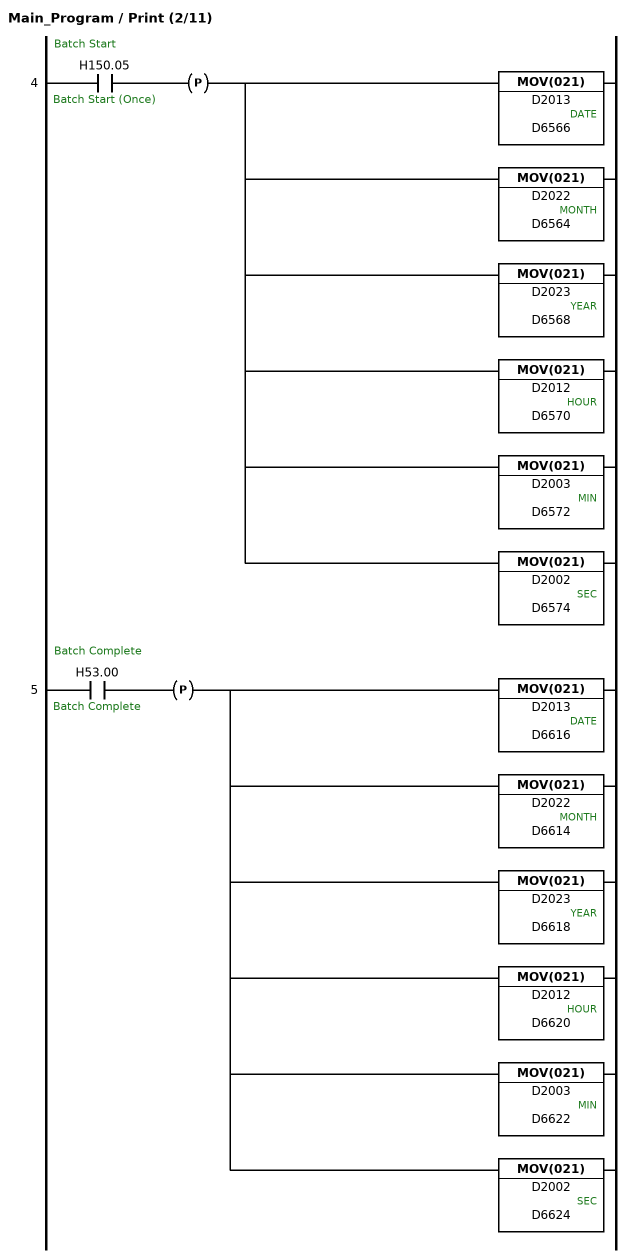
; [picture p48: Main_Program / Print, rungs 4-5]
; rung 4: Batch Start
LD H150.05  ; Batch Start (Once)
UP(521)
MOV(021) D2013 D6566  ; DATE
MOV(021) D2022 D6564  ; MONTH
MOV(021) D2023 D6568  ; YEAR
MOV(021) D2012 D6570  ; HOUR
MOV(021) D2003 D6572  ; MIN
MOV(021) D2002 D6574  ; SEC
; rung 5: Batch Complete
LD H53.00  ; Batch Complete
UP(521)
MOV(021) D2013 D6616  ; DATE
MOV(021) D2022 D6614  ; MONTH
MOV(021) D2023 D6618  ; YEAR
MOV(021) D2012 D6620  ; HOUR
MOV(021) D2003 D6622  ; MIN
MOV(021) D2002 D6624  ; SEC

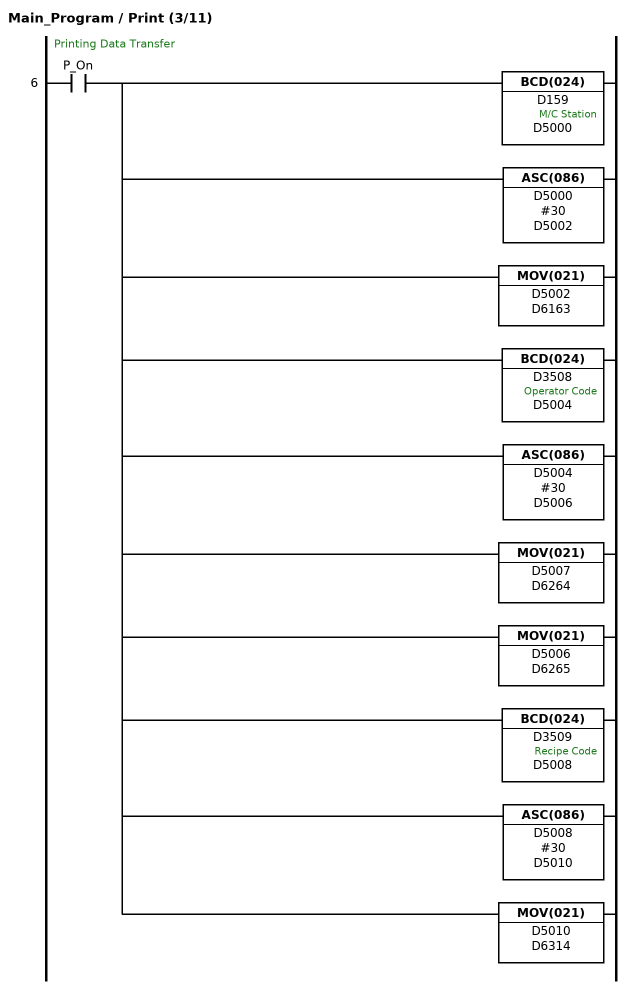
; rung 6: Printing Data Transfer
LD P_On
BCD(024) D159 D5000  ; M/C Station
ASC(086) D5000 #30 D5002
MOV(021) D5002 D6163
BCD(024) D3508 D5004  ; Operator Code
ASC(086) D5004 #30 D5006
MOV(021) D5007 D6264
MOV(021) D5006 D6265
BCD(024) D3509 D5008  ; Recipe Code
ASC(086) D5008 #30 D5010
MOV(021) D5010 D6314

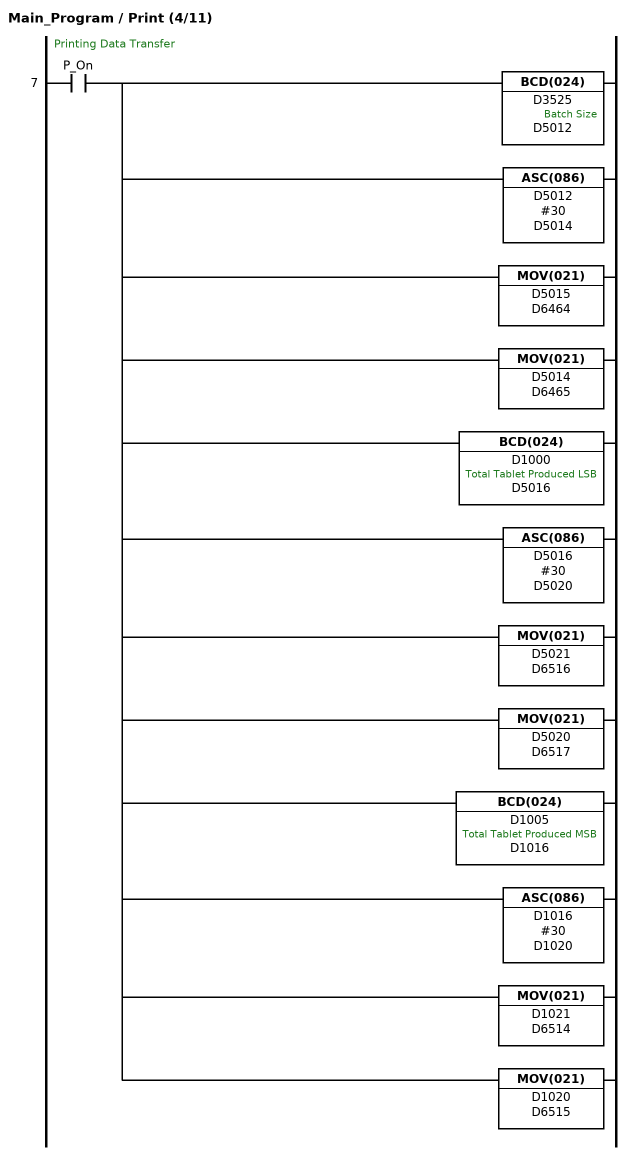
; rung 7: Printing Data Transfer
LD P_On
BCD(024) D3525 D5012  ; Batch Size
ASC(086) D5012 #30 D5014
MOV(021) D5015 D6464
MOV(021) D5014 D6465
BCD(024) D1000 D5016  ; Total Tablet Produced LSB
ASC(086) D5016 #30 D5020
MOV(021) D5021 D6516
MOV(021) D5020 D6517
BCD(024) D1005 D1016  ; Total Tablet Produced MSB
ASC(086) D1016 #30 D1020
MOV(021) D1021 D6514
MOV(021) D1020 D6515

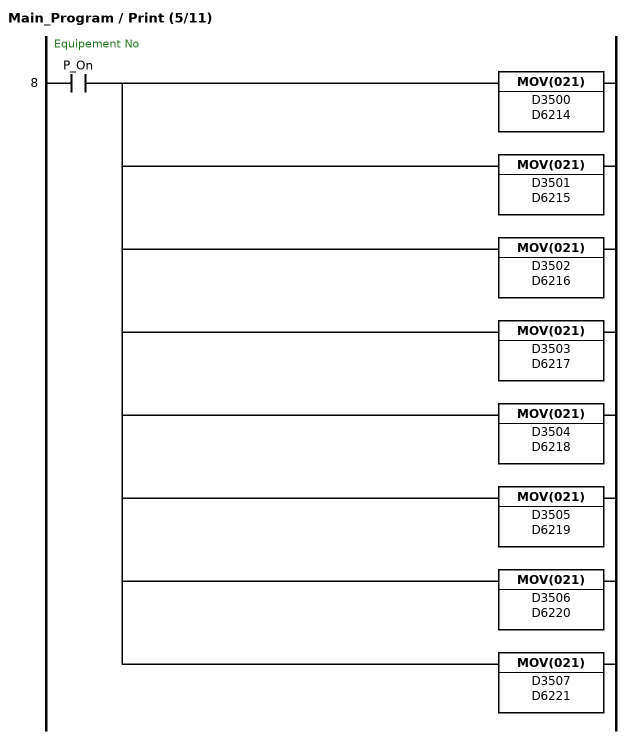
; rung 8: Equipement No
LD P_On
MOV(021) D3500 D6214
MOV(021) D3501 D6215
MOV(021) D3502 D6216
MOV(021) D3503 D6217
MOV(021) D3504 D6218
MOV(021) D3505 D6219
MOV(021) D3506 D6220
MOV(021) D3507 D6221

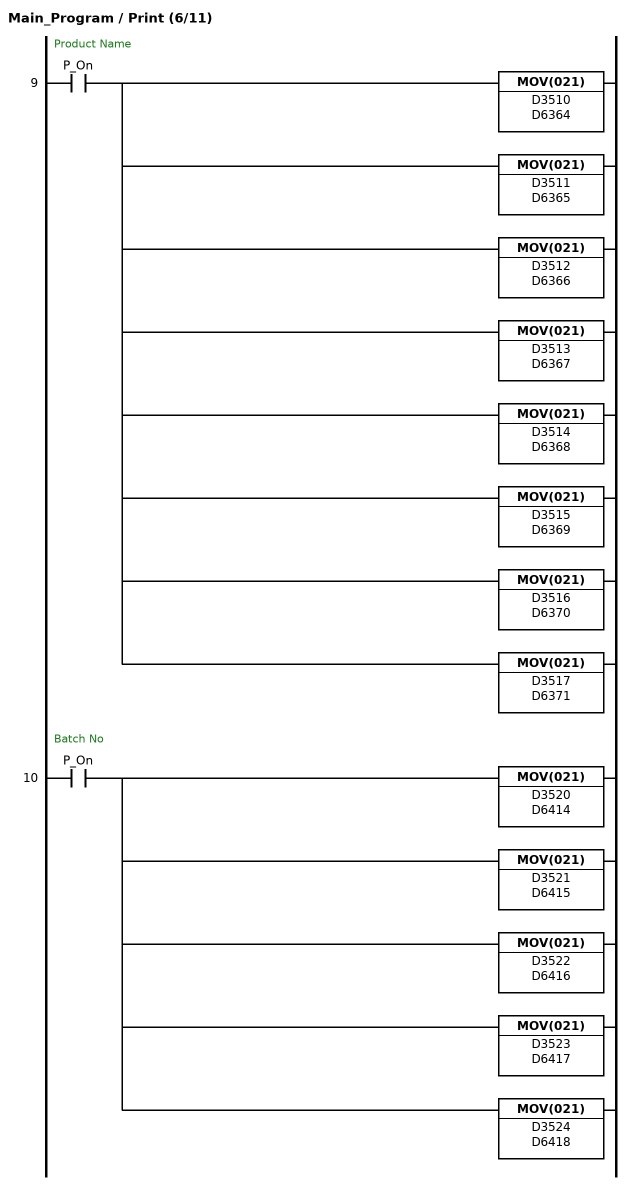
; rung 9: Product Name
LD P_On
MOV(021) D3510 D6364
MOV(021) D3511 D6365
MOV(021) D3512 D6366
MOV(021) D3513 D6367
MOV(021) D3514 D6368
MOV(021) D3515 D6369
MOV(021) D3516 D6370
MOV(021) D3517 D6371
; rung 10: Batch No
LD P_On
MOV(021) D3520 D6414
MOV(021) D3521 D6415
MOV(021) D3522 D6416
MOV(021) D3523 D6417
MOV(021) D3524 D6418

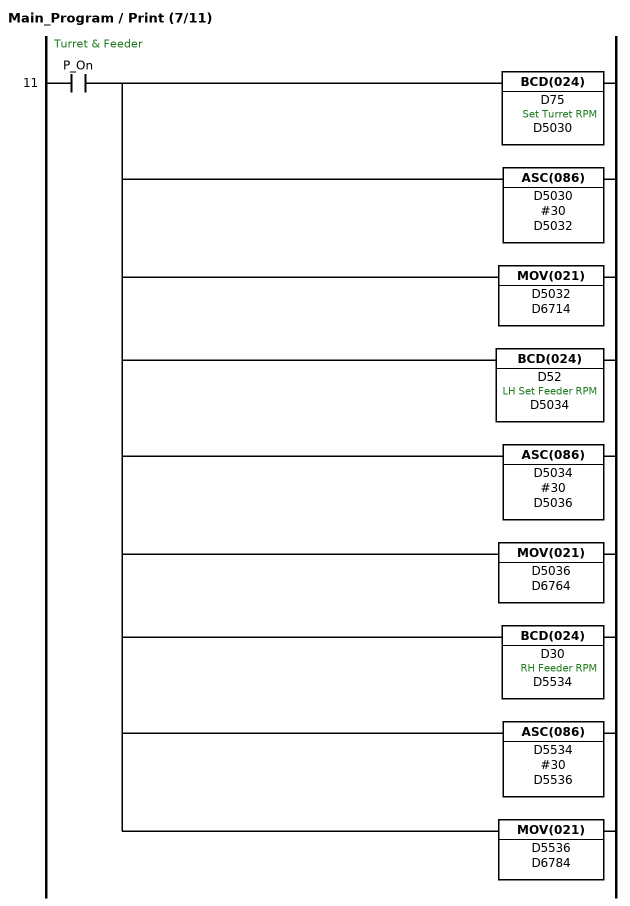
; rung 11: Turret & Feeder
LD P_On
BCD(024) D75 D5030  ; Set Turret RPM
ASC(086) D5030 #30 D5032
MOV(021) D5032 D6714
BCD(024) D52 D5034  ; LH Set Feeder RPM
ASC(086) D5034 #30 D5036
MOV(021) D5036 D6764
BCD(024) D30 D5534  ; RH Feeder RPM
ASC(086) D5534 #30 D5536
MOV(021) D5536 D6784

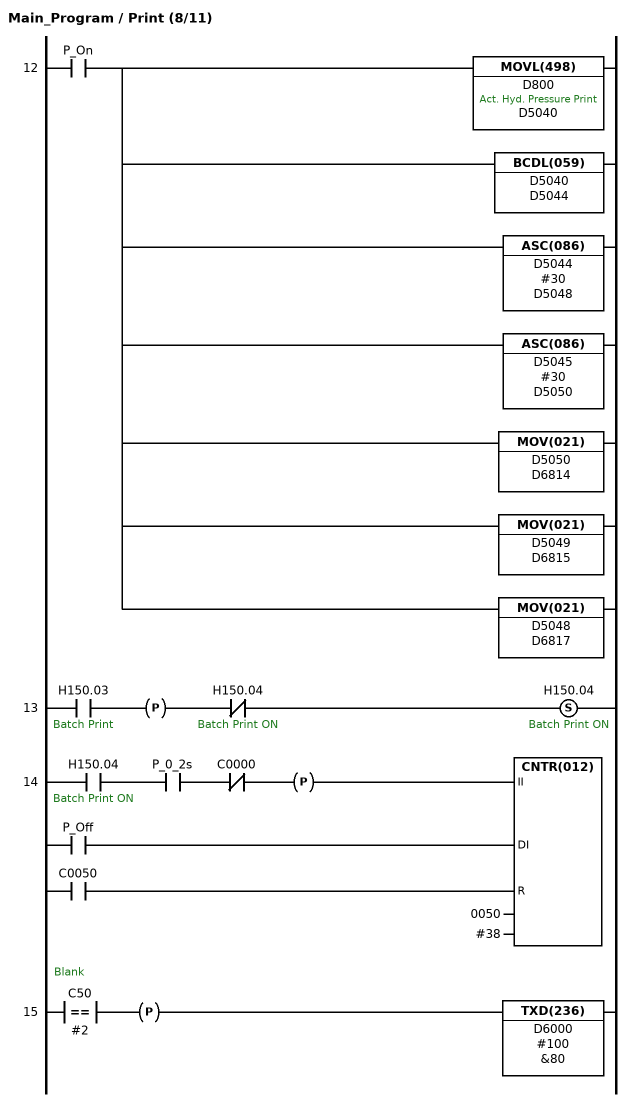
; rung 12
LD P_On
MOVL(498) D800 D5040  ; Act. Hyd. Pressure Print
BCDL(059) D5040 D5044
ASC(086) D5044 #30 D5048
ASC(086) D5045 #30 D5050
MOV(021) D5050 D6814
MOV(021) D5049 D6815
MOV(021) D5048 D6817
; rung 13
LD H150.03  ; Batch Print
UP(521)
ANDNOT H150.04  ; Batch Print ON
SET H150.04  ; Batch Print ON
; rung 14
LD H150.04  ; Batch Print ON
AND P_0_2s
ANDNOT C0000
UP(521)
LD P_Off
LD C0050
CNTR(012) 0050 #38
; rung 15: Blank
LD=(300) C50 #2
UP(521)
TXD(236) D6000 #100 &80

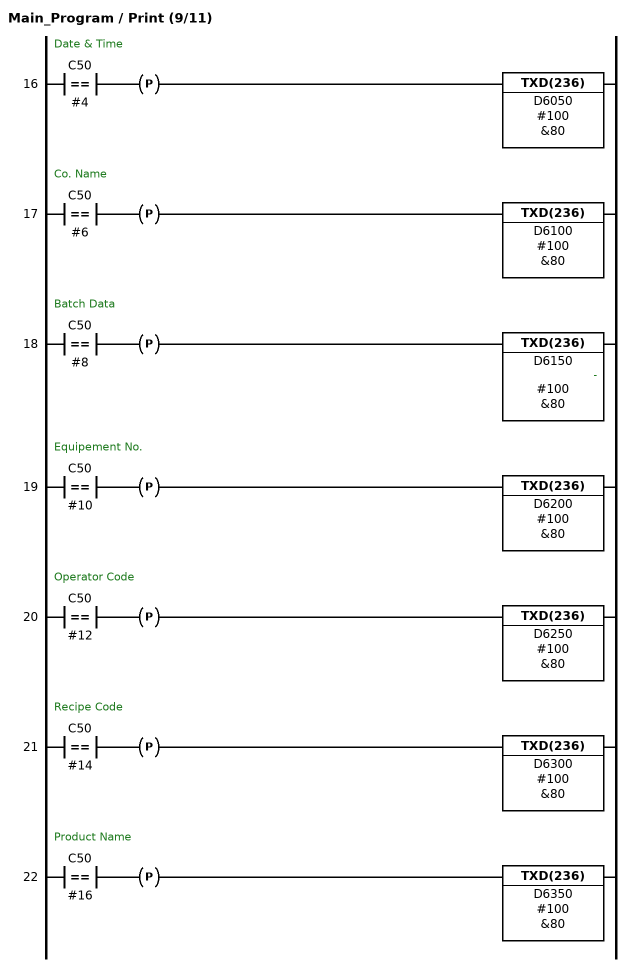
; rung 16: Date & Time
LD=(300) C50 #4
UP(521)
TXD(236) D6050 #100 &80
; rung 17: Co. Name
LD=(300) C50 #6
UP(521)
TXD(236) D6100 #100 &80
; rung 18: Batch Data
LD=(300) C50 #8
UP(521)
TXD(236) D6150 #100 &80  ; -
; rung 19: Equipement No.
LD=(300) C50 #10
UP(521)
TXD(236) D6200 #100 &80
; rung 20: Operator Code
LD=(300) C50 #12
UP(521)
TXD(236) D6250 #100 &80
; rung 21: Recipe Code
LD=(300) C50 #14
UP(521)
TXD(236) D6300 #100 &80
; rung 22: Product Name
LD=(300) C50 #16
UP(521)
TXD(236) D6350 #100 &80

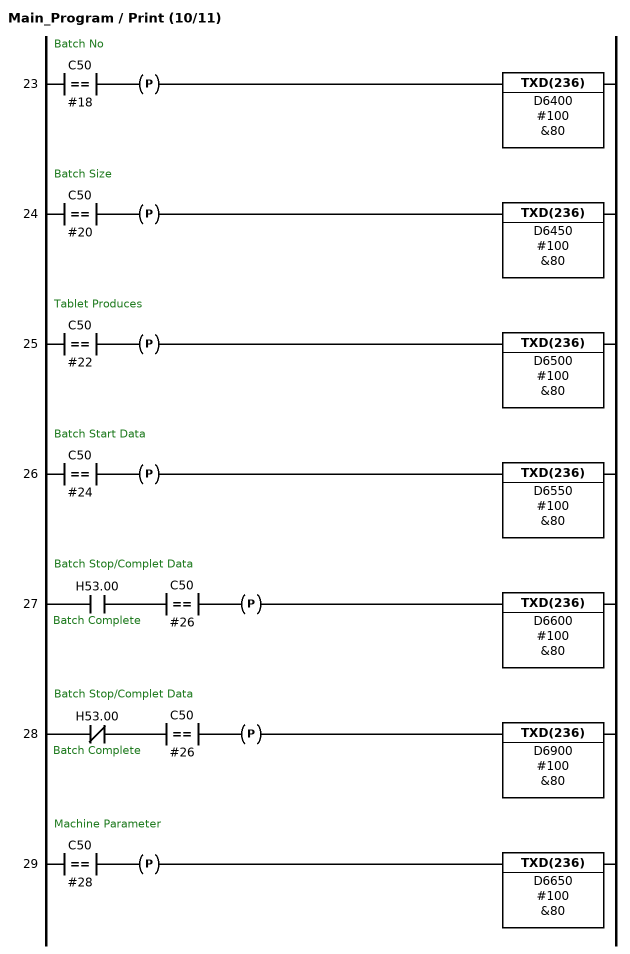
; rung 23: Batch No
LD=(300) C50 #18
UP(521)
TXD(236) D6400 #100 &80
; rung 24: Batch Size
LD=(300) C50 #20
UP(521)
TXD(236) D6450 #100 &80
; rung 25: Tablet Produces
LD=(300) C50 #22
UP(521)
TXD(236) D6500 #100 &80
; rung 26: Batch Start Data
LD=(300) C50 #24
UP(521)
TXD(236) D6550 #100 &80
; rung 27: Batch Stop/Complet Data
LD H53.00  ; Batch Complete
AND=(300) C50 #26
UP(521)
TXD(236) D6600 #100 &80
; rung 28: Batch Stop/Complet Data
LDNOT H53.00  ; Batch Complete
AND=(300) C50 #26
UP(521)
TXD(236) D6900 #100 &80
; rung 29: Machine Parameter
LD=(300) C50 #28
UP(521)
TXD(236) D6650 #100 &80

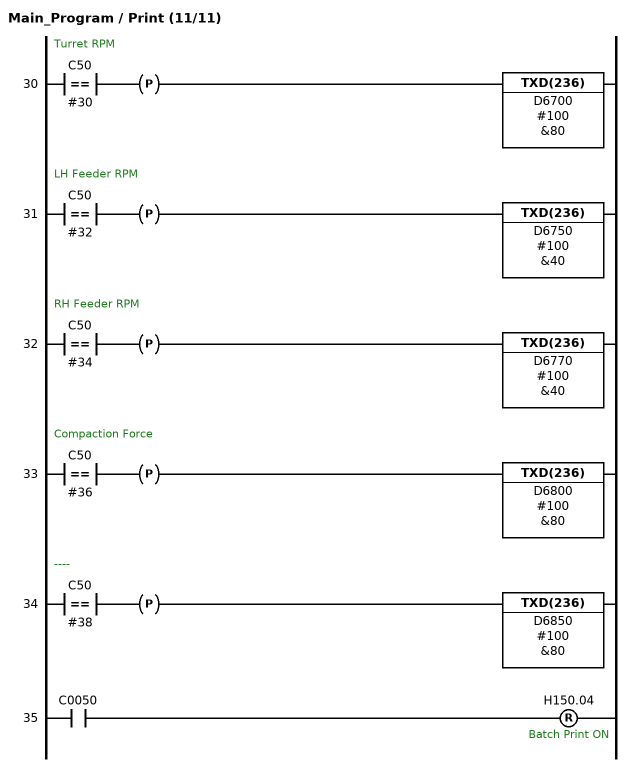
; rung 30: Turret RPM
LD=(300) C50 #30
UP(521)
TXD(236) D6700 #100 &80
; rung 31: LH Feeder RPM
LD=(300) C50 #32
UP(521)
TXD(236) D6750 #100 &40
; rung 32: RH Feeder RPM
LD=(300) C50 #34
UP(521)
TXD(236) D6770 #100 &40
; rung 33: Compaction Force
LD=(300) C50 #36
UP(521)
TXD(236) D6800 #100 &80
; rung 34: ----
LD=(300) C50 #38
UP(521)
TXD(236) D6850 #100 &80
; rung 35
LD C0050
RSET H150.04  ; Batch Print ON

### Section sampling_hooter

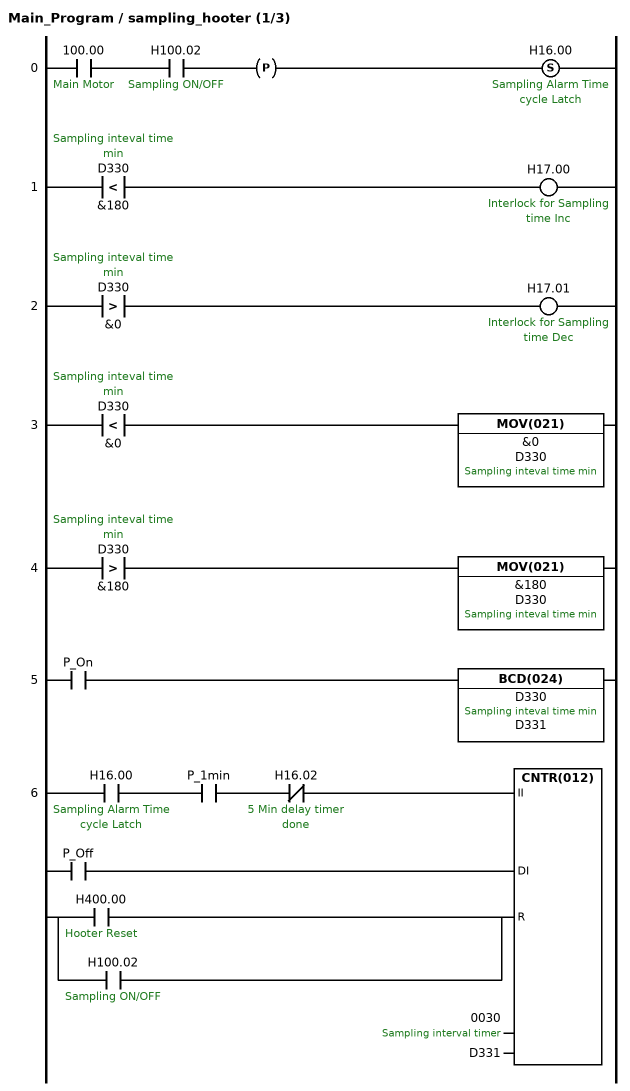
; rung 0
LD 100.00  ; Main Motor
AND H100.02  ; Sampling ON/OFF
UP(521)
SET H16.00  ; Sampling Alarm Time cycle Latch
; rung 1
LD<(310) D330 &180  ; Sampling inteval time min
OUT H17.00  ; Interlock for Sampling time Inc
; rung 2
LD>(320) D330 &0  ; Sampling inteval time min
OUT H17.01  ; Interlock for Sampling time Dec
; rung 3
LD<(310) D330 &0  ; Sampling inteval time min
MOV(021) &0 D330  ; Sampling inteval time min
; rung 4
LD>(320) D330 &180  ; Sampling inteval time min
MOV(021) &180 D330  ; Sampling inteval time min
; rung 5
LD P_On
BCD(024) D330 D331  ; Sampling inteval time min
; rung 6
LD H16.00  ; Sampling Alarm Time cycle Latch
AND P_1min
ANDNOT H16.02  ; 5 Min delay timer done
LD P_Off
LD H400.00  ; Hooter Reset
OR H100.02  ; Sampling ON/OFF
CNTR(012) 0030 D331  ; Sampling interval timer

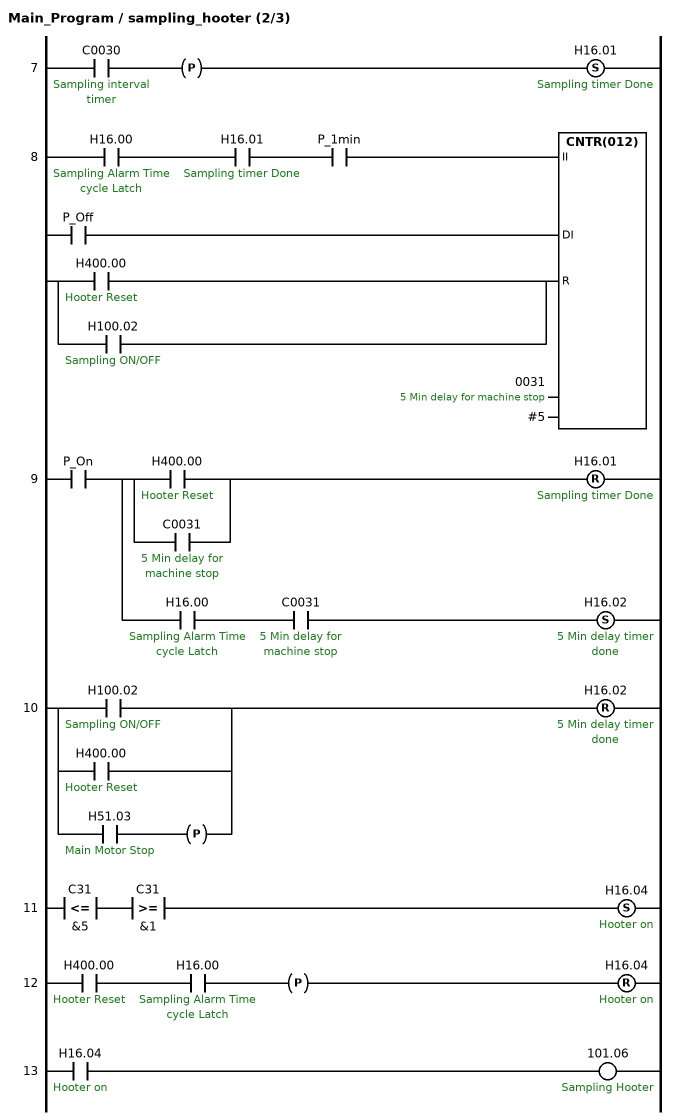
; rung 7
LD C0030  ; Sampling interval timer
UP(521)
SET H16.01  ; Sampling timer Done
; rung 8
LD H16.00  ; Sampling Alarm Time cycle Latch
AND H16.01  ; Sampling timer Done
AND P_1min
LD P_Off
LD H400.00  ; Hooter Reset
OR H100.02  ; Sampling ON/OFF
CNTR(012) 0031 #5  ; 5 Min delay for machine stop
; rung 9
LD P_On
OUT TR0
LD H400.00  ; Hooter Reset
OR C0031  ; 5 Min delay for machine stop
ANDLD
RSET H16.01  ; Sampling timer Done
LD TR0
AND H16.00  ; Sampling Alarm Time cycle Latch
AND C0031  ; 5 Min delay for machine stop
SET H16.02  ; 5 Min delay timer done
; rung 10
LD H100.02  ; Sampling ON/OFF
OR H400.00  ; Hooter Reset
LD H51.03  ; Main Motor Stop
UP(521)
ORLD
RSET H16.02  ; 5 Min delay timer done
; rung 11
LD<=(315) C31 &5
AND>=(325) C31 &1
SET H16.04  ; Hooter on
; rung 12
LD H400.00  ; Hooter Reset
AND H16.00  ; Sampling Alarm Time cycle Latch
UP(521)
RSET H16.04  ; Hooter on
; rung 13
LD H16.04  ; Hooter on
OUT 101.06  ; Sampling Hooter

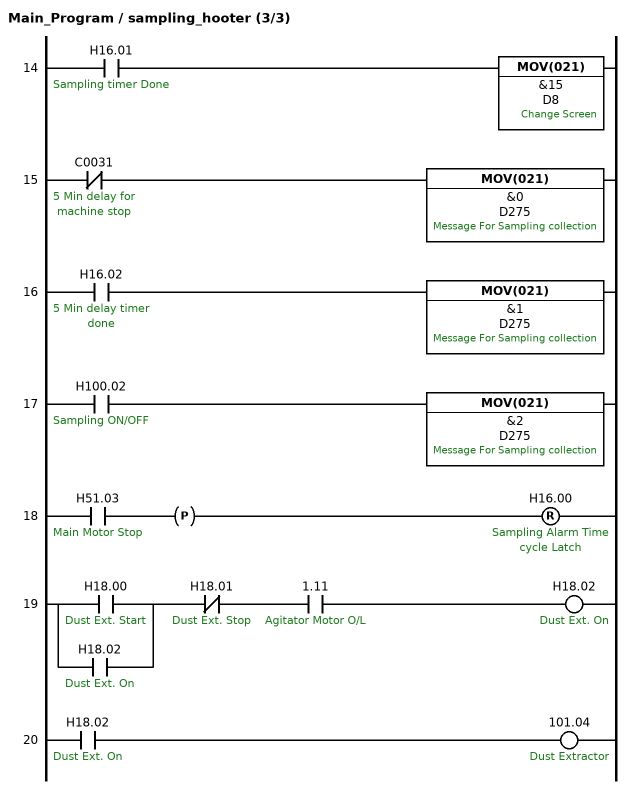
; rung 14
LD H16.01  ; Sampling timer Done
MOV(021) &15 D8  ; Change Screen
; rung 15
LDNOT C0031  ; 5 Min delay for machine stop
MOV(021) &0 D275  ; Message For Sampling collection
; rung 16
LD H16.02  ; 5 Min delay timer done
MOV(021) &1 D275  ; Message For Sampling collection
; rung 17
LD H100.02  ; Sampling ON/OFF
MOV(021) &2 D275  ; Message For Sampling collection
; rung 18
LD H51.03  ; Main Motor Stop
UP(521)
RSET H16.00  ; Sampling Alarm Time cycle Latch
; rung 19
LD H18.00  ; Dust Ext. Start
OR H18.02  ; Dust Ext. On
ANDNOT H18.01  ; Dust Ext. Stop
AND 1.11  ; Agitator Motor O/L
OUT H18.02  ; Dust Ext. On
; rung 20
LD H18.02  ; Dust Ext. On
OUT 101.04  ; Dust Extractor

### Section Vac_U_Max

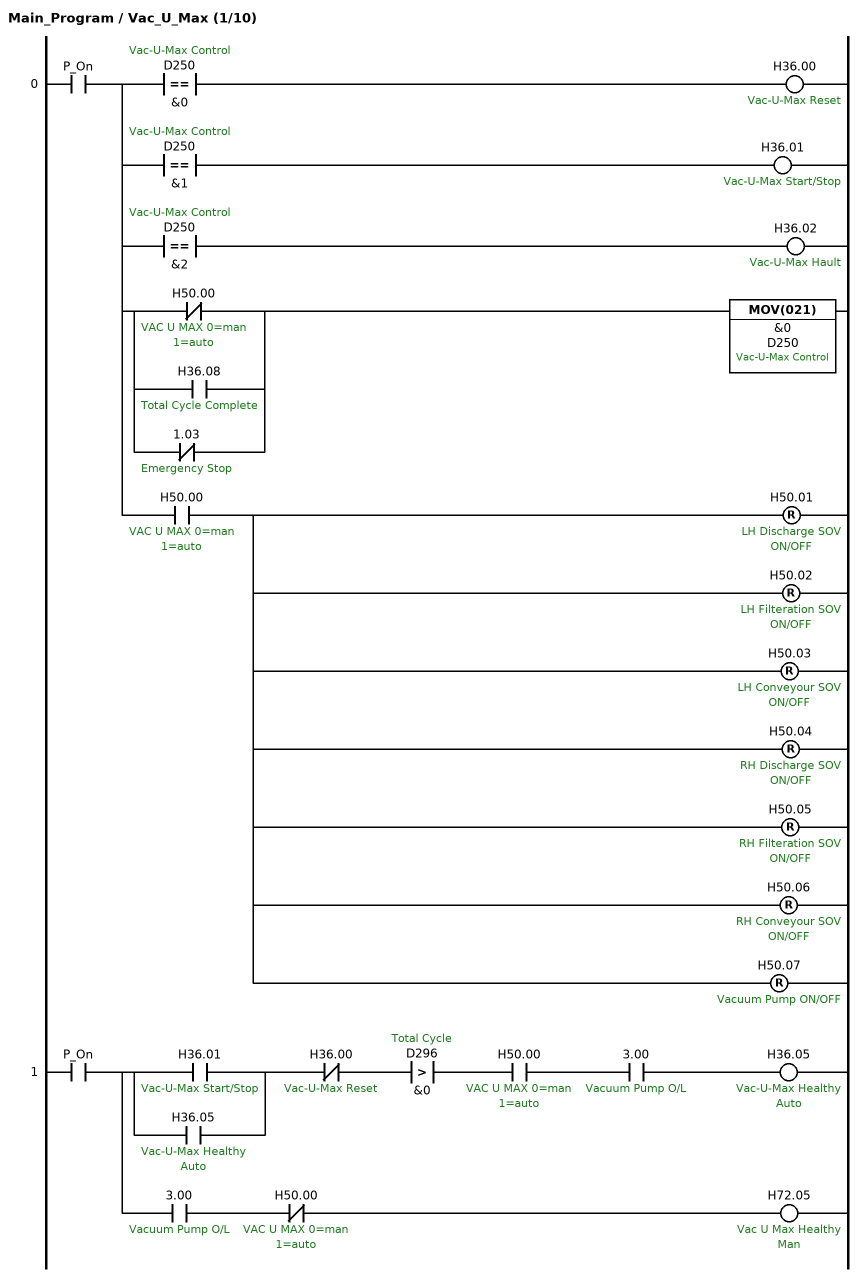
; rung 0
LD P_On
OUT TR0
AND=(300) D250 &0  ; Vac-U-Max Control
OUT H36.00  ; Vac-U-Max Reset
LD TR0
AND=(300) D250 &1  ; Vac-U-Max Control
OUT H36.01  ; Vac-U-Max Start/Stop
LD TR0
AND=(300) D250 &2  ; Vac-U-Max Control
OUT H36.02  ; Vac-U-Max Hault
LD TR0
LDNOT H50.00  ; VAC U MAX 0=man 1=auto
OR H36.08  ; Total Cycle Complete
ORNOT 1.03  ; Emergency Stop
ANDLD
MOV(021) &0 D250  ; Vac-U-Max Control
LD TR0
AND H50.00  ; VAC U MAX 0=man 1=auto
RSET H50.01  ; LH Discharge SOV ON/OFF
RSET H50.02  ; LH Filteration SOV ON/OFF
RSET H50.03  ; LH Conveyour SOV ON/OFF
RSET H50.04  ; RH Discharge SOV ON/OFF
RSET H50.05  ; RH Filteration SOV ON/OFF
RSET H50.06  ; RH Conveyour SOV ON/OFF
RSET H50.07  ; Vacuum Pump ON/OFF
; rung 1
LD P_On
OUT TR0
LD H36.01  ; Vac-U-Max Start/Stop
OR H36.05  ; Vac-U-Max Healthy Auto
ANDLD
ANDNOT H36.00  ; Vac-U-Max Reset
AND>(320) D296 &0  ; Total Cycle
AND H50.00  ; VAC U MAX 0=man 1=auto
AND 3.00  ; Vacuum Pump O/L
OUT H36.05  ; Vac-U-Max Healthy Auto
LD TR0
AND 3.00  ; Vacuum Pump O/L
ANDNOT H50.00  ; VAC U MAX 0=man 1=auto
OUT H72.05  ; Vac U Max Healthy Man

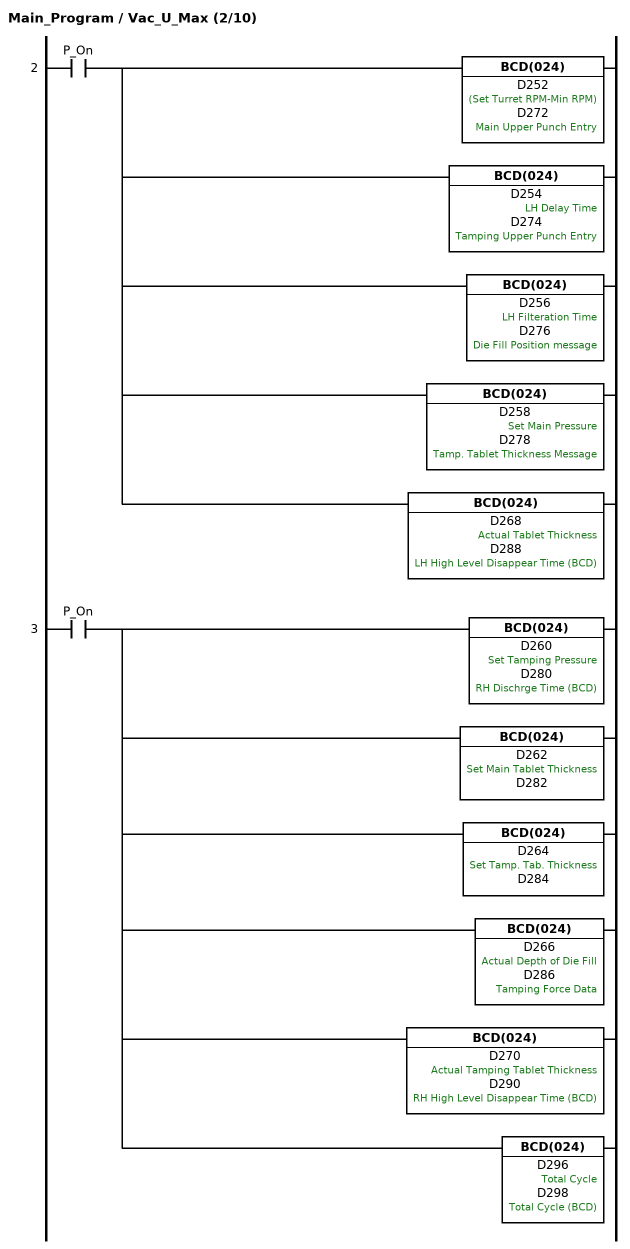
; rung 2
LD P_On
BCD(024) D252 D272  ; (Set Turret RPM-Min RPM), Main Upper Punch Entry
BCD(024) D254 D274  ; LH Delay Time, Tamping Upper Punch Entry
BCD(024) D256 D276  ; LH Filteration Time, Die Fill Position message
BCD(024) D258 D278  ; Set Main Pressure, Tamp. Tablet Thickness Message
BCD(024) D268 D288  ; Actual Tablet Thickness, LH High Level Disappear Time (BCD)
; rung 3
LD P_On
BCD(024) D260 D280  ; Set Tamping Pressure, RH Dischrge Time (BCD)
BCD(024) D262 D282  ; Set Main Tablet Thickness
BCD(024) D264 D284  ; Set Tamp. Tab. Thickness
BCD(024) D266 D286  ; Actual Depth of Die Fill, Tamping Force Data
BCD(024) D270 D290  ; Actual Tamping Tablet Thickness, RH High Level Disappear Time (BCD)
BCD(024) D296 D298  ; Total Cycle, Total Cycle (BCD)

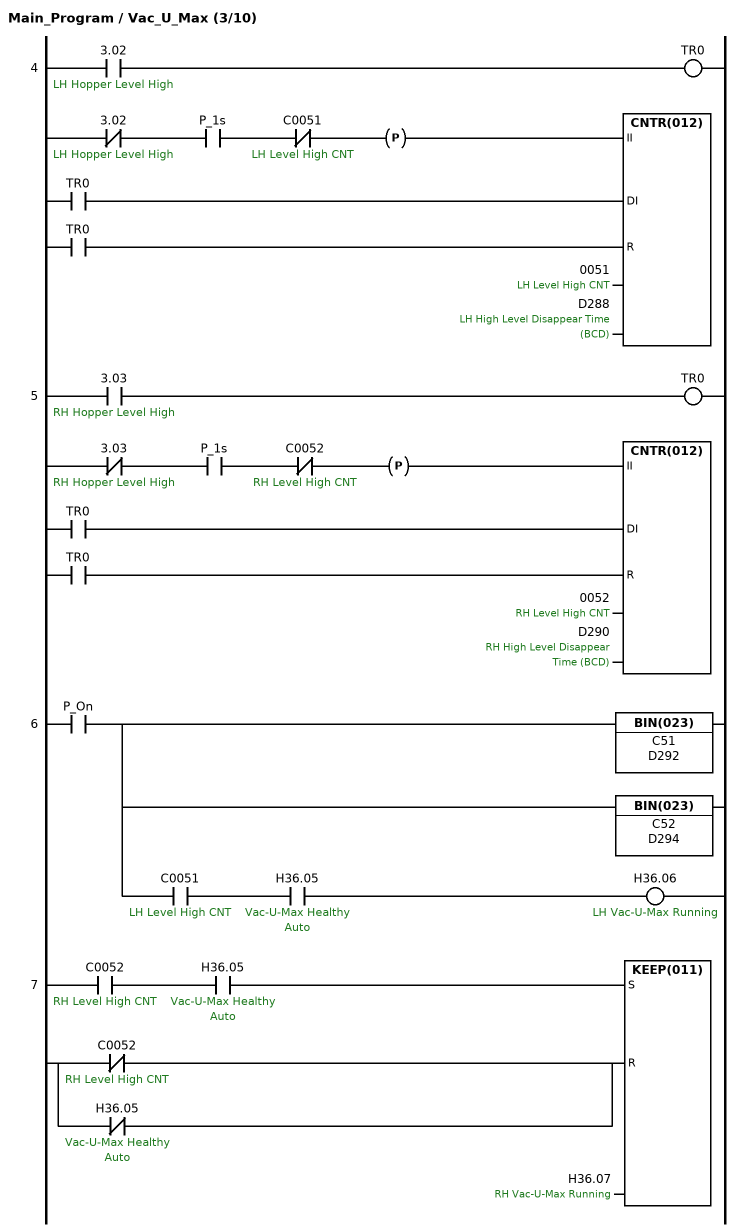
; rung 4
LDNOT 3.02  ; LH Hopper Level High
AND P_1s
ANDNOT C0051  ; LH Level High CNT
UP(521)
LD 3.02  ; LH Hopper Level High
OUT TR0
LD TR0
CNTR(012) 0051 D288  ; LH High Level Disappear Time (BCD), LH Level High CNT
; rung 5
LDNOT 3.03  ; RH Hopper Level High
AND P_1s
ANDNOT C0052  ; RH Level High CNT
UP(521)
LD 3.03  ; RH Hopper Level High
OUT TR0
LD TR0
CNTR(012) 0052 D290  ; RH High Level Disappear Time (BCD), RH Level High CNT
; rung 6
LD P_On
BIN(023) C51 D292
BIN(023) C52 D294
AND C0051  ; LH Level High CNT
AND H36.05  ; Vac-U-Max Healthy Auto
OUT H36.06  ; LH Vac-U-Max Running
; rung 7
LD C0052  ; RH Level High CNT
AND H36.05  ; Vac-U-Max Healthy Auto
LDNOT C0052  ; RH Level High CNT
ORNOT H36.05  ; Vac-U-Max Healthy Auto
KEEP(011) H36.07  ; RH Vac-U-Max Running

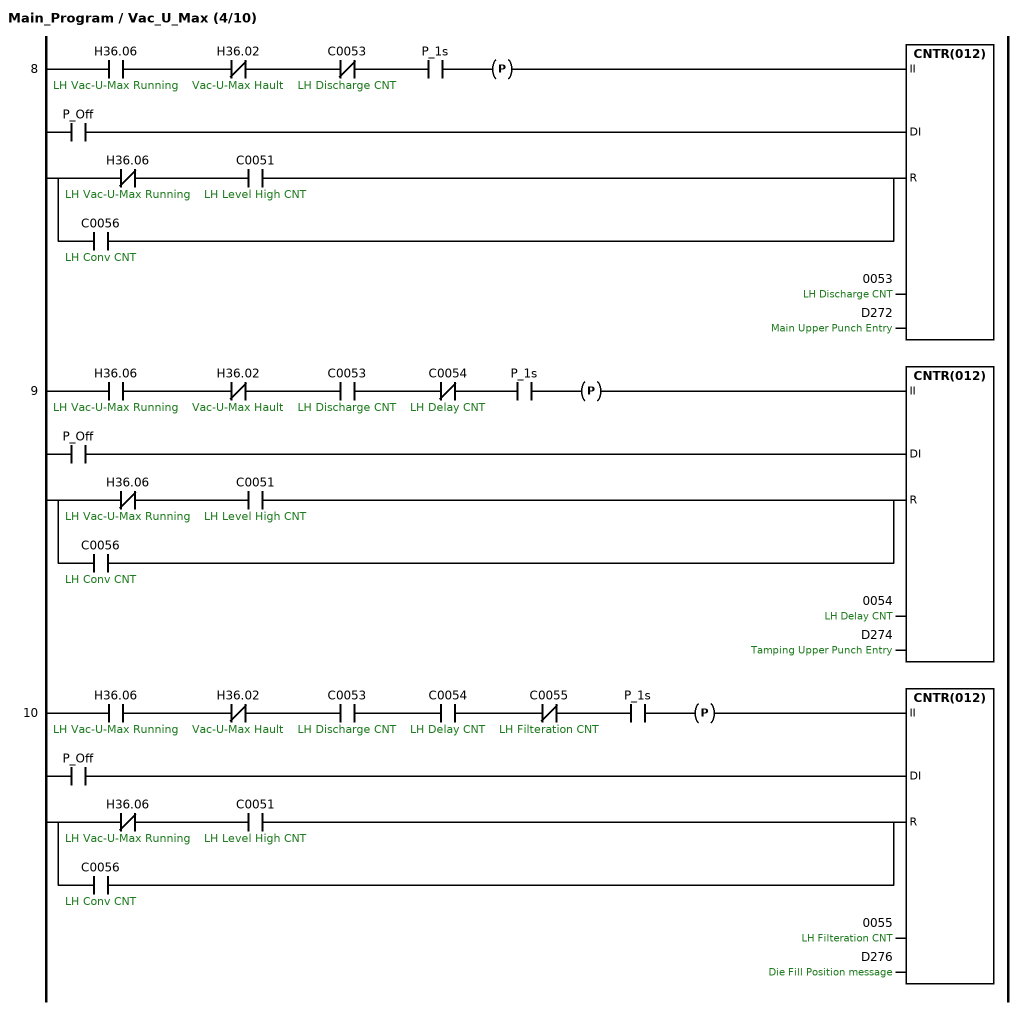
; rung 8
LD H36.06  ; LH Vac-U-Max Running
ANDNOT H36.02  ; Vac-U-Max Hault
ANDNOT C0053  ; LH Discharge CNT
AND P_1s
UP(521)
LD P_Off
LDNOT H36.06  ; LH Vac-U-Max Running
AND C0051  ; LH Level High CNT
OR C0056  ; LH Conv CNT
CNTR(012) 0053 D272  ; Main Upper Punch Entry, LH Discharge CNT
; rung 9
LD H36.06  ; LH Vac-U-Max Running
ANDNOT H36.02  ; Vac-U-Max Hault
AND C0053  ; LH Discharge CNT
ANDNOT C0054  ; LH Delay CNT
AND P_1s
UP(521)
LD P_Off
LDNOT H36.06  ; LH Vac-U-Max Running
AND C0051  ; LH Level High CNT
OR C0056  ; LH Conv CNT
CNTR(012) 0054 D274  ; Tamping Upper Punch Entry, LH Delay CNT
; rung 10
LD H36.06  ; LH Vac-U-Max Running
ANDNOT H36.02  ; Vac-U-Max Hault
AND C0053  ; LH Discharge CNT
AND C0054  ; LH Delay CNT
ANDNOT C0055  ; LH Filteration CNT
AND P_1s
UP(521)
LD P_Off
LDNOT H36.06  ; LH Vac-U-Max Running
AND C0051  ; LH Level High CNT
OR C0056  ; LH Conv CNT
CNTR(012) 0055 D276  ; Die Fill Position message, LH Filteration CNT

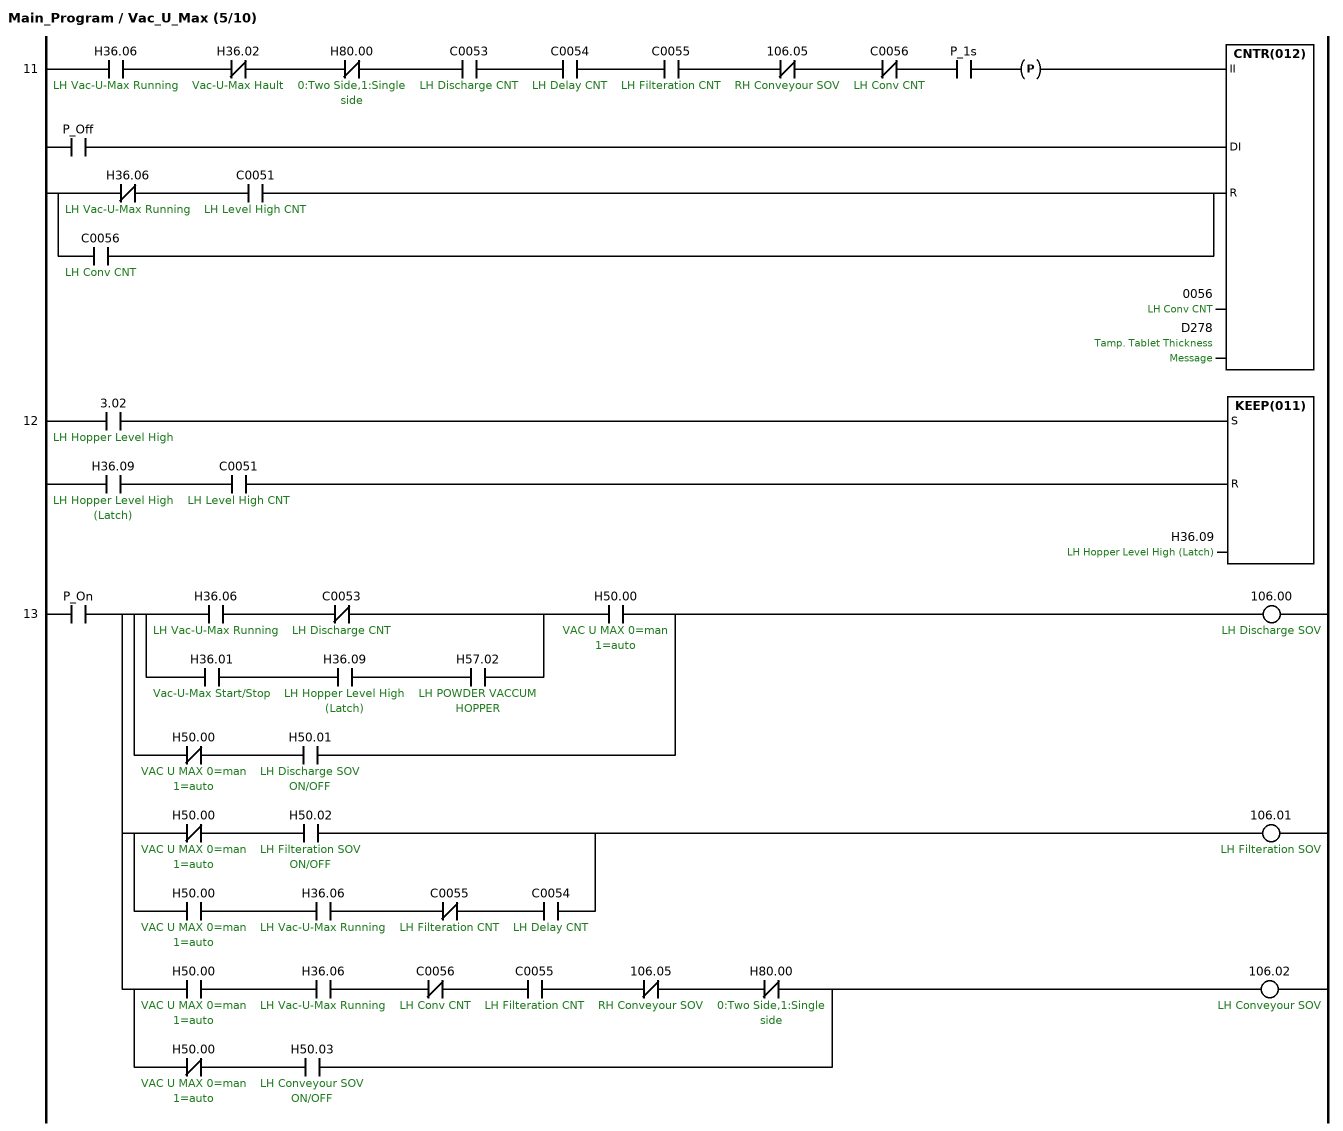
; rung 11
LD H36.06  ; LH Vac-U-Max Running
ANDNOT H36.02  ; Vac-U-Max Hault
ANDNOT H80.00  ; 0:Two Side,1:Single side
AND C0053  ; LH Discharge CNT
AND C0054  ; LH Delay CNT
AND C0055  ; LH Filteration CNT
ANDNOT 106.05  ; RH Conveyour SOV
ANDNOT C0056  ; LH Conv CNT
AND P_1s
UP(521)
LD P_Off
LDNOT H36.06  ; LH Vac-U-Max Running
AND C0051  ; LH Level High CNT
OR C0056  ; LH Conv CNT
CNTR(012) 0056 D278  ; Tamp. Tablet Thickness Message, LH Conv CNT
; rung 12
LD 3.02  ; LH Hopper Level High
LD H36.09  ; LH Hopper Level High (Latch)
AND C0051  ; LH Level High CNT
KEEP(011) H36.09  ; LH Hopper Level High (Latch)
; rung 13
LD P_On
OUT TR0
LD H36.06  ; LH Vac-U-Max Running
ANDNOT C0053  ; LH Discharge CNT
LD H36.01  ; Vac-U-Max Start/Stop
AND H36.09  ; LH Hopper Level High (Latch)
AND H57.02  ; LH POWDER VACCUM HOPPER
ORLD
AND H50.00  ; VAC U MAX 0=man 1=auto
LDNOT H50.00  ; VAC U MAX 0=man 1=auto
AND H50.01  ; LH Discharge SOV ON/OFF
ORLD
ANDLD
OUT 106.00  ; LH Discharge SOV
LD TR0
LDNOT H50.00  ; VAC U MAX 0=man 1=auto
AND H50.02  ; LH Filteration SOV ON/OFF
LD H50.00  ; VAC U MAX 0=man 1=auto
AND H36.06  ; LH Vac-U-Max Running
ANDNOT C0055  ; LH Filteration CNT
AND C0054  ; LH Delay CNT
ORLD
ANDLD
OUT 106.01  ; LH Filteration SOV
LD TR0
LD H50.00  ; VAC U MAX 0=man 1=auto
AND H36.06  ; LH Vac-U-Max Running
ANDNOT C0056  ; LH Conv CNT
AND C0055  ; LH Filteration CNT
ANDNOT 106.05  ; RH Conveyour SOV
ANDNOT H80.00  ; 0:Two Side,1:Single side
LDNOT H50.00  ; VAC U MAX 0=man 1=auto
AND H50.03  ; LH Conveyour SOV ON/OFF
ORLD
ANDLD
OUT 106.02  ; LH Conveyour SOV

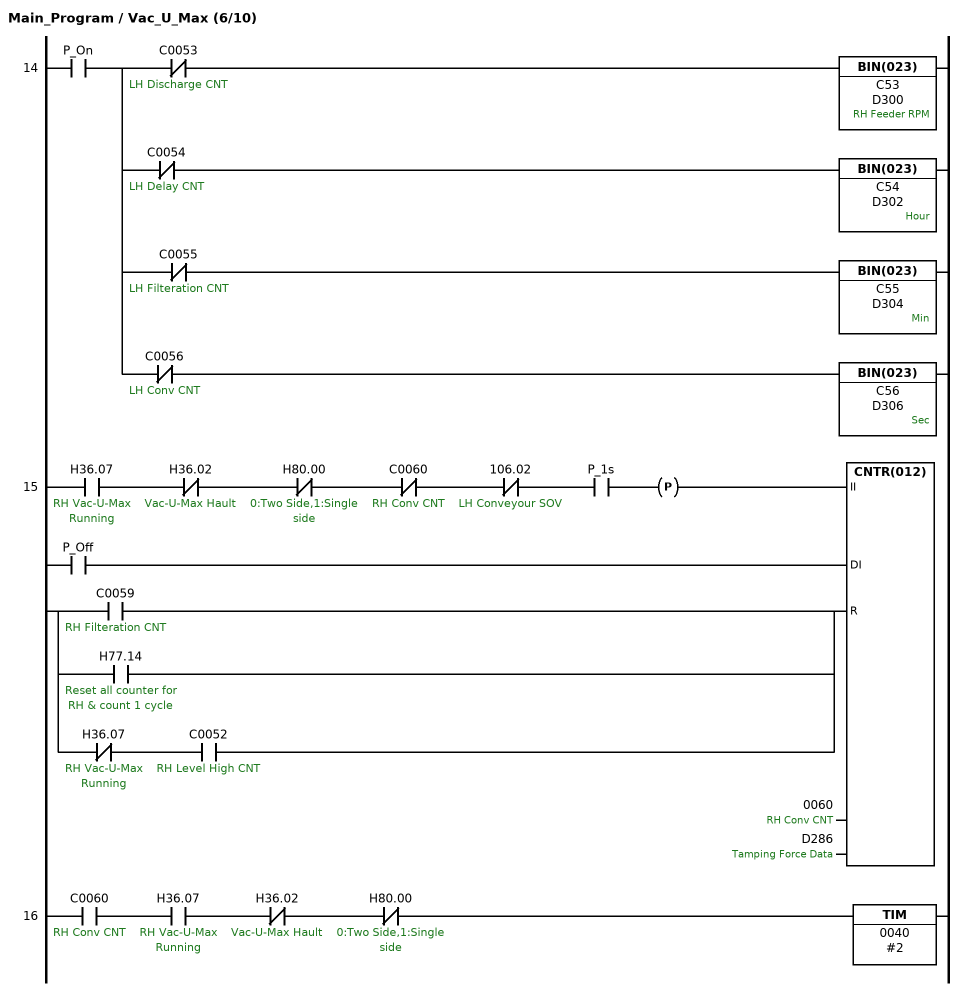
; rung 14
LD P_On
OUT TR0
ANDNOT C0053  ; LH Discharge CNT
BIN(023) C53 D300  ; RH Feeder RPM
LD TR0
ANDNOT C0054  ; LH Delay CNT
BIN(023) C54 D302  ; Hour
LD TR0
ANDNOT C0055  ; LH Filteration CNT
BIN(023) C55 D304  ; Min
LD TR0
ANDNOT C0056  ; LH Conv CNT
BIN(023) C56 D306  ; Sec
; rung 15
LD H36.07  ; RH Vac-U-Max Running
ANDNOT H36.02  ; Vac-U-Max Hault
ANDNOT H80.00  ; 0:Two Side,1:Single side
ANDNOT C0060  ; RH Conv CNT
ANDNOT 106.02  ; LH Conveyour SOV
AND P_1s
UP(521)
LD P_Off
LD C0059  ; RH Filteration CNT
OR H77.14  ; Reset all counter for RH & count 1 cycle
LDNOT H36.07  ; RH Vac-U-Max Running
AND C0052  ; RH Level High CNT
ORLD
CNTR(012) 0060 D286  ; Tamping Force Data, RH Conv CNT
; rung 16
LD C0060  ; RH Conv CNT
AND H36.07  ; RH Vac-U-Max Running
ANDNOT H36.02  ; Vac-U-Max Hault
ANDNOT H80.00  ; 0:Two Side,1:Single side
TIM 0040 #2

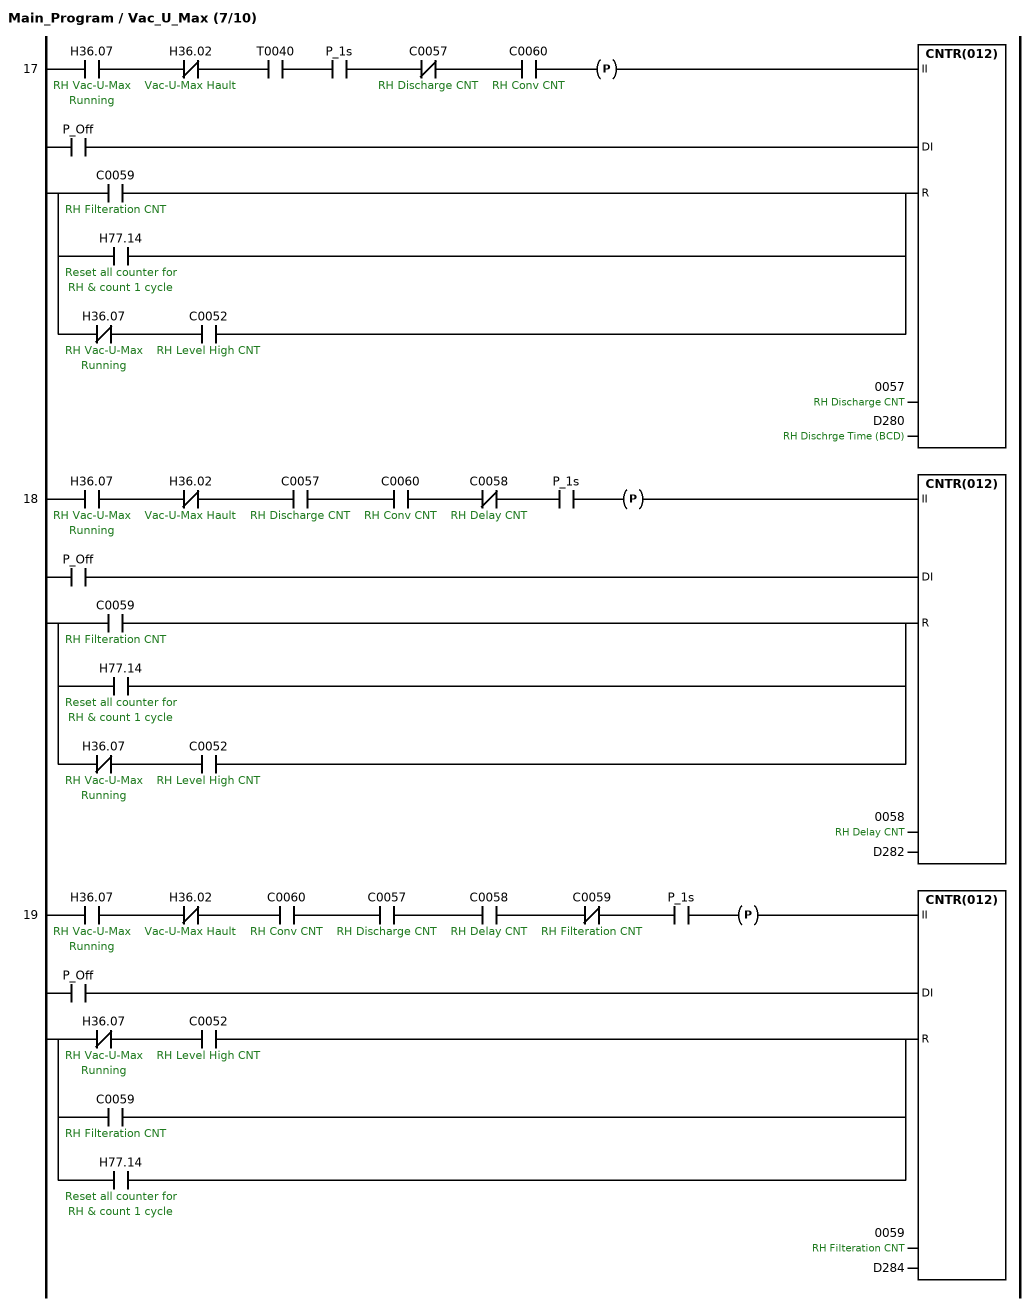
; rung 17
LD H36.07  ; RH Vac-U-Max Running
ANDNOT H36.02  ; Vac-U-Max Hault
AND T0040
AND P_1s
ANDNOT C0057  ; RH Discharge CNT
AND C0060  ; RH Conv CNT
UP(521)
LD P_Off
LD C0059  ; RH Filteration CNT
OR H77.14  ; Reset all counter for RH & count 1 cycle
LDNOT H36.07  ; RH Vac-U-Max Running
AND C0052  ; RH Level High CNT
ORLD
CNTR(012) 0057 D280  ; RH Dischrge Time (BCD), RH Discharge CNT
; rung 18
LD H36.07  ; RH Vac-U-Max Running
ANDNOT H36.02  ; Vac-U-Max Hault
AND C0057  ; RH Discharge CNT
AND C0060  ; RH Conv CNT
ANDNOT C0058  ; RH Delay CNT
AND P_1s
UP(521)
LD P_Off
LD C0059  ; RH Filteration CNT
OR H77.14  ; Reset all counter for RH & count 1 cycle
LDNOT H36.07  ; RH Vac-U-Max Running
AND C0052  ; RH Level High CNT
ORLD
CNTR(012) 0058 D282  ; RH Delay CNT
; rung 19
LD H36.07  ; RH Vac-U-Max Running
ANDNOT H36.02  ; Vac-U-Max Hault
AND C0060  ; RH Conv CNT
AND C0057  ; RH Discharge CNT
AND C0058  ; RH Delay CNT
ANDNOT C0059  ; RH Filteration CNT
AND P_1s
UP(521)
LD P_Off
LDNOT H36.07  ; RH Vac-U-Max Running
AND C0052  ; RH Level High CNT
OR C0059  ; RH Filteration CNT
OR H77.14  ; Reset all counter for RH & count 1 cycle
CNTR(012) 0059 D284  ; RH Filteration CNT

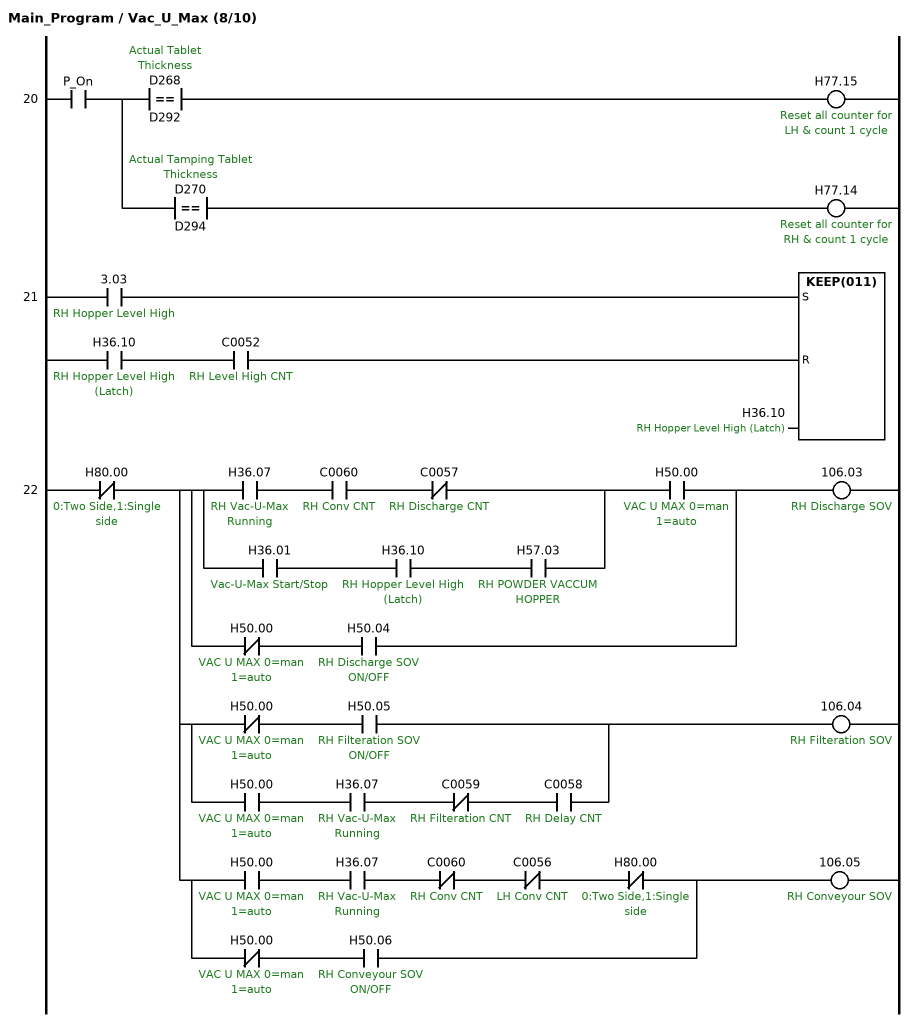
; rung 20
LD P_On
OUT TR0
AND=(300) D268 D292  ; Actual Tablet Thickness
OUT H77.15  ; Reset all counter for LH & count 1 cycle
LD TR0
AND=(300) D270 D294  ; Actual Tamping Tablet Thickness
OUT H77.14  ; Reset all counter for RH & count 1 cycle
; rung 21
LD 3.03  ; RH Hopper Level High
LD H36.10  ; RH Hopper Level High (Latch)
AND C0052  ; RH Level High CNT
KEEP(011) H36.10  ; RH Hopper Level High (Latch)
; rung 22
LDNOT H80.00  ; 0:Two Side,1:Single side
OUT TR0
LD H36.07  ; RH Vac-U-Max Running
AND C0060  ; RH Conv CNT
ANDNOT C0057  ; RH Discharge CNT
LD H36.01  ; Vac-U-Max Start/Stop
AND H36.10  ; RH Hopper Level High (Latch)
AND H57.03  ; RH POWDER VACCUM HOPPER
ORLD
AND H50.00  ; VAC U MAX 0=man 1=auto
LDNOT H50.00  ; VAC U MAX 0=man 1=auto
AND H50.04  ; RH Discharge SOV ON/OFF
ORLD
ANDLD
OUT 106.03  ; RH Discharge SOV
LD TR0
LDNOT H50.00  ; VAC U MAX 0=man 1=auto
AND H50.05  ; RH Filteration SOV ON/OFF
LD H50.00  ; VAC U MAX 0=man 1=auto
AND H36.07  ; RH Vac-U-Max Running
ANDNOT C0059  ; RH Filteration CNT
AND C0058  ; RH Delay CNT
ORLD
ANDLD
OUT 106.04  ; RH Filteration SOV
LD TR0
LD H50.00  ; VAC U MAX 0=man 1=auto
AND H36.07  ; RH Vac-U-Max Running
ANDNOT C0060  ; RH Conv CNT
ANDNOT C0056  ; LH Conv CNT
ANDNOT H80.00  ; 0:Two Side,1:Single side
LDNOT H50.00  ; VAC U MAX 0=man 1=auto
AND H50.06  ; RH Conveyour SOV ON/OFF
ORLD
ANDLD
OUT 106.05  ; RH Conveyour SOV

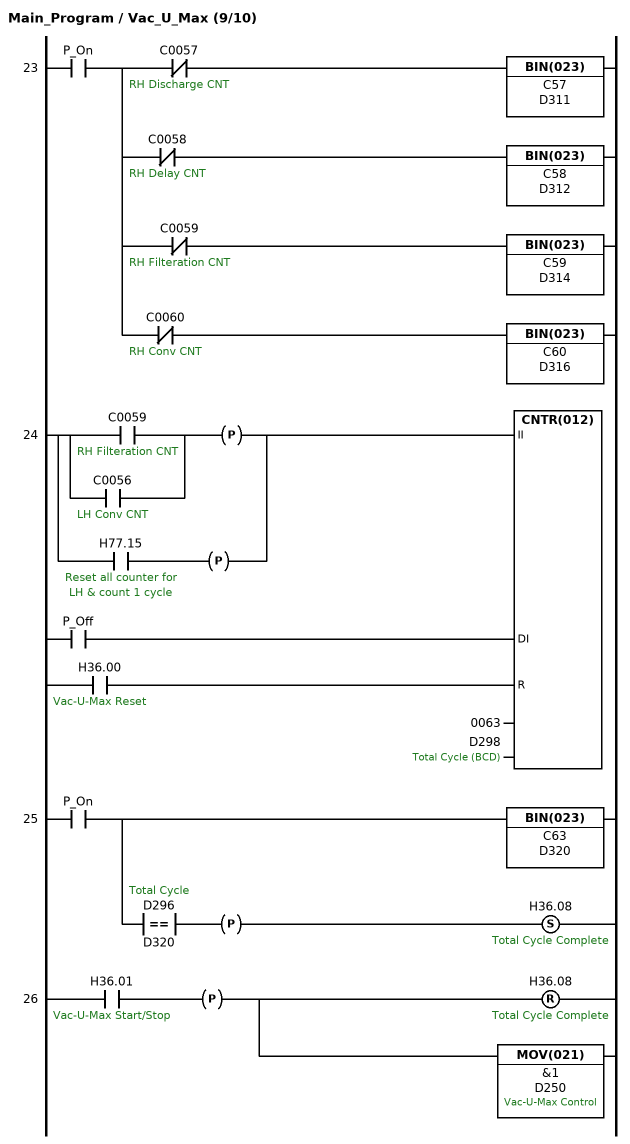
; rung 23
LD P_On
OUT TR0
ANDNOT C0057  ; RH Discharge CNT
BIN(023) C57 D311
LD TR0
ANDNOT C0058  ; RH Delay CNT
BIN(023) C58 D312
LD TR0
ANDNOT C0059  ; RH Filteration CNT
BIN(023) C59 D314
LD TR0
ANDNOT C0060  ; RH Conv CNT
BIN(023) C60 D316
; rung 24
LD C0059  ; RH Filteration CNT
OR C0056  ; LH Conv CNT
UP(521)
LD H77.15  ; Reset all counter for LH & count 1 cycle
UP(521)
ORLD
LD P_Off
LD H36.00  ; Vac-U-Max Reset
CNTR(012) 0063 D298  ; Total Cycle (BCD)
; rung 25
LD P_On
BIN(023) C63 D320
AND=(300) D296 D320  ; Total Cycle
UP(521)
SET H36.08  ; Total Cycle Complete
; rung 26
LD H36.01  ; Vac-U-Max Start/Stop
UP(521)
RSET H36.08  ; Total Cycle Complete
MOV(021) &1 D250  ; Vac-U-Max Control

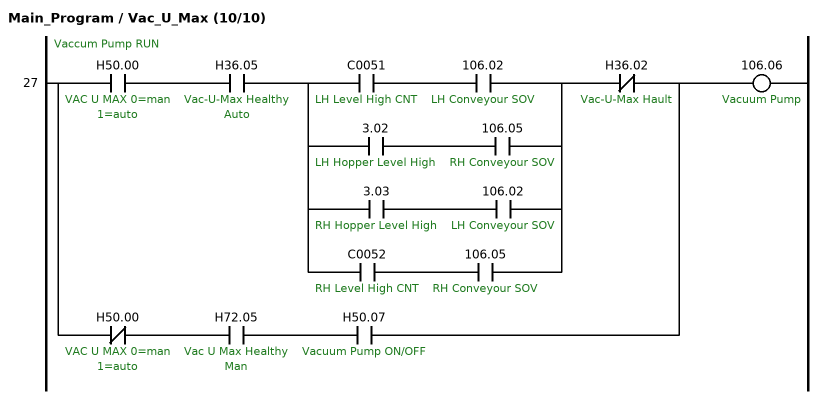
; rung 27: Vaccum Pump RUN
LD H50.00  ; VAC U MAX 0=man 1=auto
AND H36.05  ; Vac-U-Max Healthy Auto
LD C0051  ; LH Level High CNT
AND 106.02  ; LH Conveyour SOV
LD 3.02  ; LH Hopper Level High
AND 106.05  ; RH Conveyour SOV
ORLD
LD 3.03  ; RH Hopper Level High
AND 106.02  ; LH Conveyour SOV
ORLD
LD C0052  ; RH Level High CNT
AND 106.05  ; RH Conveyour SOV
ORLD
ANDLD
ANDNOT H36.02  ; Vac-U-Max Hault
LDNOT H50.00  ; VAC U MAX 0=man 1=auto
AND H72.05  ; Vac U Max Healthy Man
AND H50.07  ; Vacuum Pump ON/OFF
ORLD
OUT 106.06  ; Vacuum Pump

### Section END
; rung 0
END(001)

## Function block FRTC
VAR_INPUT
  MNSC : INT;
  DTHR : INT;
  YRMN : INT;
END_VAR
VAR_OUTPUT
  OHR : INT;
  OMIN : INT;
  OSEC : INT;
  ODT : INT;
  OMN : INT;
  OYR : INT;
END_VAR
VAR
  DMNSC : INT;
  OMNSC : ARRAY[0..1] OF INT;
  DDTHR : INT;
  ODTHR : ARRAY[0..1] OF INT;
  DYRMN : INT;
  OYRMN : ARRAY[0..1] OF INT;
END_VAR

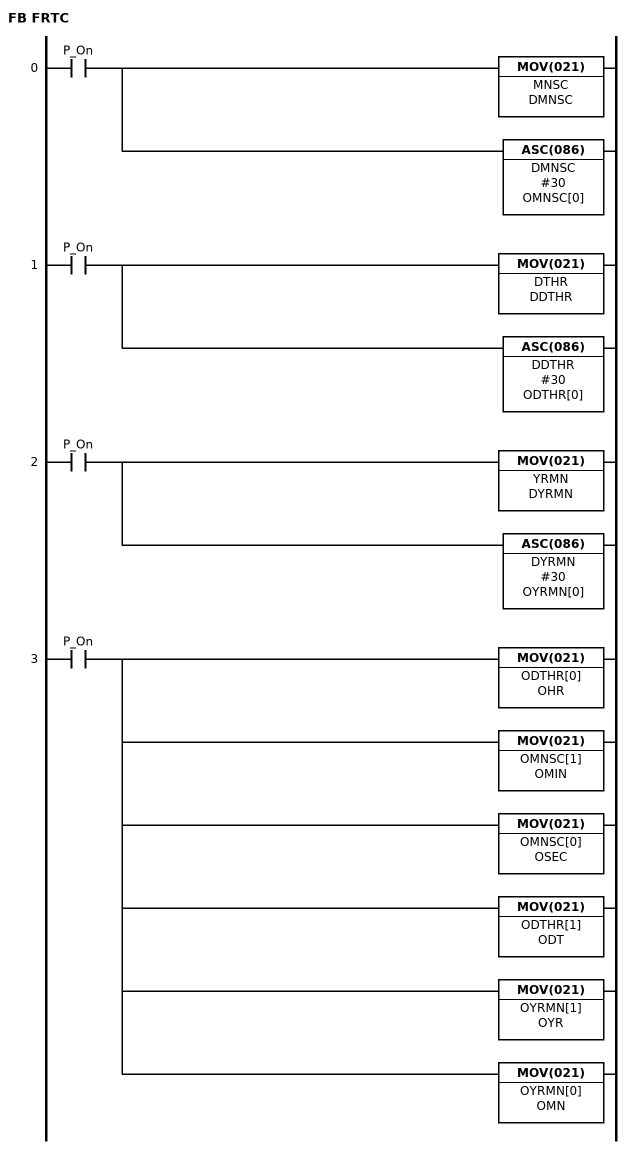
; rung 0
LD P_On
MOV(021) MNSC DMNSC
ASC(086) DMNSC #30 OMNSC[0]
; rung 1
LD P_On
MOV(021) DTHR DDTHR
ASC(086) DDTHR #30 ODTHR[0]
; rung 2
LD P_On
MOV(021) YRMN DYRMN
ASC(086) DYRMN #30 OYRMN[0]
; rung 3
LD P_On
MOV(021) ODTHR[0] OHR
MOV(021) OMNSC[1] OMIN
MOV(021) OMNSC[0] OSEC
MOV(021) ODTHR[1] ODT
MOV(021) OYRMN[1] OYR
MOV(021) OYRMN[0] OMN

## Function block SCP
VAR_INPUT
  Scal_max : REAL;
  Scal_min : REAL;
  Input_max : REAL;
  Input_min : REAL;
  Input : INT;
END_VAR
VAR_OUTPUT
  Output : INT;
END_VAR
VAR
  IP_Real : REAL;
  OP_R : REAL;
END_VAR
IP_Real := Int_to_Real(Input);
OP_R := (((Scal_max-Scal_min)/(Input_max-Input_min))*(IP_Real-Input_min))+Scal_min ;
Output := Real_to_Int(OP_R);

## Function block SCP_Hyd
VAR_INPUT
  Scal_max : REAL;
  Scal_min : REAL;
  Input_max : REAL;
  Input_min : REAL;
  Input : INT;
END_VAR
VAR_OUTPUT
  Output : INT;
END_VAR
VAR
  IP_Real : REAL;
  OP_R : REAL;
END_VAR
IP_Real := Int_to_Real(Input);
IF Int_to_Real( Input) < Input_min THEN;
      IP_Real:= Input_min;
END_IF;

OP_R := (((Scal_max-Scal_min)/(Input_max-Input_min))*(IP_Real-Input_min))+Scal_min ;
Output := Real_to_Int(OP_R);